SUBAPPLICATION Uebung_010a3_AX (* Button_L1 (Latching) auf DigitalOutput_Q1 *)
  (* Standard: 61499-2; Description: Copyright (c) 2023 Meisterschulen am Ostbahnhof This program and the accompanying materials are made available under the terms of the Eclipse Public License 2.0 which is available at https://www.eclipse.org/legal/epl-2.0/ SPDX-License-Identifier: EPL-2.0 *)
  (* Version 1.0, 2026-01-14, Franz Höpfinger, Meisterschulen am Ostbahnhof, initial API and implementation and/or initial documentation *)
  PACKAGE Uebungen;
  IMPORT Uebungen::const::UT::DefaultPool::Button_L1;
  IMPORT logiBUS::io::DQ::logiBUS_DO::Output_Q1;
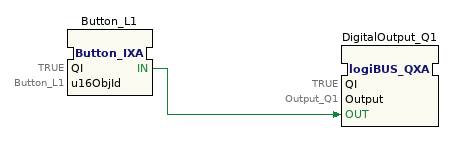
  (* Latching Button "rastet ein" kein T_FF nötig! *)
  FBS
    DigitalOutput_Q1 : logiBUS::io::DQ::logiBUS_QXA(QI := TRUE, Output := Output_Q1);
    Button_L1 : isobus::UT::io::Button::Button_IXA(QI := TRUE, u16ObjId := Button_L1);
  END_FBS
  ADAPTER_CONNECTIONS
    Button_L1.IN TO DigitalOutput_Q1.OUT;
  END_CONNECTIONS
END_SUBAPPLICATION
